TYPE ST_CoordSys :
STRUCT
    id       : DINT;
    plant_id : DINT;

    name : STRING(255);

    x : LREAL;
    y : LREAL;
    z : LREAL;

    rx : LREAL;
    ry : LREAL;
    rz : LREAL;
END_STRUCT
END_TYPE

(* stored: Version 1.1.0.1, ProductVersion 3.1.4026.18
   DUT ST_CoordSys: Id {228b6cfb-4ecb-4b34-9c8c-0f5e98b6e278} *)
